FUNCTION_BLOCK TN_INPUT_SELECT_POPUP
VAR
	in_index : INT;
	in_Element_Count : INT;
	by_Cur_Key : BYTE;
	by_Attr : BYTE;
	st_String : STRING;
END_VAR
VAR
	us_TN_MENU_POPUP : us_TN_MENU_POPUP;
	FB_TN_INPUT_MENU_POPUP : TN_INPUT_MENU_POPUP;
	FB_TN_SC_WRITE : TN_SC_WRITE;
END_VAR
VAR_IN_OUT
	Xus_TN_SCREEN : us_TN_SCREEN;
	Xus_TN_INPUT_CONTROL_DATA : us_TN_INPUT_CONTROL_DATA;
END_VAR

(*
version 1.1		06. apr 2011
programmer		ks
tested by			ks

TN_SELECT_POPUP dient zur verwaltung und darstellung eines POPUP-Dialogs zur Elementeauswahl
*)

(* Benutzereingabe auswerten -> Selektion Text n *)
IF (Xus_TN_INPUT_CONTROL_DATA.bo_Focus = TRUE) THEN

	by_Cur_Key := Xus_TN_INPUT_CONTROL_DATA.by_Input_Exten_Code;

	IF (us_TN_MENU_POPUP.bo_Activ = FALSE) THEN
		us_TN_MENU_POPUP.by_Input_Exten_Code := BYTE#00;

		(* Return-Taste auswerten *)
		IF (by_Cur_Key = BYTE#13) THEN
			(* Popup-Menu parameter übergeben *)
			us_TN_MENU_POPUP.in_Y := Xus_TN_INPUT_CONTROL_DATA.in_Y;
			us_TN_MENU_POPUP.in_X := Xus_TN_INPUT_CONTROL_DATA.in_X;
			us_TN_MENU_POPUP.by_Attr_mF := Xus_TN_INPUT_CONTROL_DATA.by_Attr_mF;
			us_TN_MENU_POPUP.by_Attr_oF := Xus_TN_INPUT_CONTROL_DATA.by_Attr_oF;
			us_TN_MENU_POPUP.st_Menu_Text := Xus_TN_INPUT_CONTROL_DATA.st_Input_Data;
			us_TN_MENU_POPUP.bo_Create := TRUE;
			us_TN_MENU_POPUP.in_Cur_Item := INT#00;
		END_IF;

		IF (us_TN_MENU_POPUP.in_Cur_Item > INT#00) THEN
			Xus_TN_INPUT_CONTROL_DATA.in_selected := us_TN_MENU_POPUP.in_Cur_Item;
			Xus_TN_INPUT_CONTROL_DATA.bo_Input_Entered := TRUE;
			Xus_TN_INPUT_CONTROL_DATA.bo_Update_Input := TRUE;
			us_TN_MENU_POPUP.in_Cur_Item := INT#00;
		END_IF;

	ELSE
		us_TN_MENU_POPUP.by_Input_Exten_Code := by_Cur_Key;
	END_IF;

	(* Popup-Menu zyklisch aufrufen *)
	FB_TN_INPUT_MENU_POPUP(Xus_TN_MENU_POPUP := us_TN_MENU_POPUP, Xus_TN_SCREEN := Xus_TN_SCREEN);

END_IF;

(* Aktualisierung der Anzeige *)
IF (Xus_TN_INPUT_CONTROL_DATA.bo_Update_Input = TRUE) OR (Xus_TN_INPUT_CONTROL_DATA.bo_Update_All = TRUE) THEN

	(* Title-Text ausgeben *)
	IF Xus_TN_INPUT_CONTROL_DATA.bo_Update_All = TRUE THEN

		IF (Xus_TN_INPUT_CONTROL_DATA.in_Title_X_Offset = INT#00) AND (Xus_TN_INPUT_CONTROL_DATA.in_Title_Y_Offset = INT#00) THEN
			(* wenn Offset X,Y =0 dann Titlestring links vom Element positionieren *)
			FB_TN_SC_WRITE.Iin_Y := Xus_TN_INPUT_CONTROL_DATA.in_Y;
			FB_TN_SC_WRITE.Iin_X := Xus_TN_INPUT_CONTROL_DATA.in_X - LEN(Xus_TN_INPUT_CONTROL_DATA.st_Title_String);

		ELSE
			(* Title-Text durch Row, Color-Offset ausgeben *)
			FB_TN_SC_WRITE.Iin_Y := Xus_TN_INPUT_CONTROL_DATA.in_Y + Xus_TN_INPUT_CONTROL_DATA.in_Title_Y_Offset;
			FB_TN_SC_WRITE.Iin_X := Xus_TN_INPUT_CONTROL_DATA.in_X + Xus_TN_INPUT_CONTROL_DATA.in_Title_X_Offset;
		END_IF;

		(* Title-Text durch Row, Color-Offset ausgeben *)
		FB_TN_SC_WRITE(	Iby_ATTR := Xus_TN_INPUT_CONTROL_DATA.by_Title_Attr,
						Ist_STRING := Xus_TN_INPUT_CONTROL_DATA.st_Title_String,
						Xus_TN_SCREEN := Xus_TN_SCREEN);
	END_IF;

	in_Element_Count := ELEMENT_COUNT(SEP:=BYTE#35,ELEMENT:=Xus_TN_INPUT_CONTROL_DATA.st_Input_Data);

	IF in_Element_Count > INT#00 THEN

		Xus_TN_INPUT_CONTROL_DATA.in_selected:=LIMIT(1,Xus_TN_INPUT_CONTROL_DATA.in_selected,in_Element_Count);

		in_index := Xus_TN_INPUT_CONTROL_DATA.in_selected;

		st_String := ELEMENT_GET(SEP:=BYTE#35,POS:=in_index - 1,ELEMENT:=Xus_TN_INPUT_CONTROL_DATA.st_Input_Data);

		st_String:= FIX(str:=st_String,
						L:=LEN(Xus_TN_INPUT_CONTROL_DATA.st_Input_Mask),
						C:=BYTE#32,
						M:=Xus_TN_INPUT_CONTROL_DATA.in_Input_Option);


		Xus_TN_INPUT_CONTROL_DATA.st_Input_String := st_String;

		IF Xus_TN_INPUT_CONTROL_DATA.bo_Focus = TRUE THEN
			by_Attr := Xus_TN_INPUT_CONTROL_DATA.by_Attr_mF;
		ELSE
			by_Attr := Xus_TN_INPUT_CONTROL_DATA.by_Attr_oF;
		END_IF;

		FB_TN_SC_WRITE(	Iin_X := Xus_TN_INPUT_CONTROL_DATA.in_X,
								Iin_Y := Xus_TN_INPUT_CONTROL_DATA.in_Y,
								Iby_ATTR := by_Attr,
								Ist_STRING := st_String,
								Xus_TN_SCREEN := Xus_TN_SCREEN );
	END_IF;

	(* Cursor auf aktuelle Position setzen *)
	Xus_TN_INPUT_CONTROL_DATA.in_Cursor_X := Xus_TN_INPUT_CONTROL_DATA.in_X;
	Xus_TN_INPUT_CONTROL_DATA.in_Cursor_Y := Xus_TN_INPUT_CONTROL_DATA.in_Y;

	(* Update-Flag's rücksetzen *)
	Xus_TN_INPUT_CONTROL_DATA.bo_Update_All   := FALSE;
	Xus_TN_INPUT_CONTROL_DATA.bo_Update_Input := FALSE;

END_IF;

(* revision history

ks	06. apr. 2011	rev 1.1
	list_len und list_get durch element_count und element_get ersetzt

ks	10. mai. 2010	rev 1.0
	original version
*)

END_FUNCTION_BLOCK

(* stored: Version 1.1.0.1, ProductVersion 3.1.4024.0
   POU TN_INPUT_SELECT_POPUP: Id {6f3d1917-8b7d-47b9-8a01-7102e7156887}, SpecialFunc None *)
